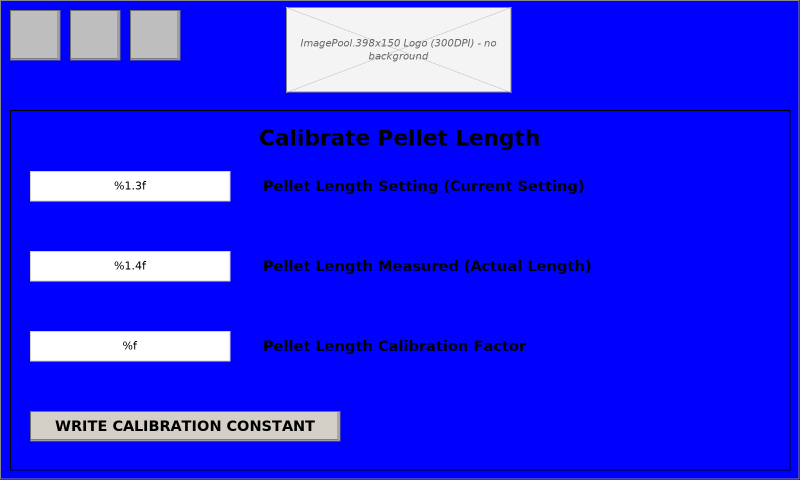
VISUALIZATION Calibrate_Settings  // 800x480
    Rectangle (0,0 800x480)
    Rectangle (10,110 780x360)
    Textfield (30,171 200x30), "%1.3f", text variable: GVL.Pellet_Length_Inch_Input
    Textfield (30,251 200x30), "%1.4f", text variable: Pellet_Calibration.Pellet_Length_Measured_Input
        OnMouseClick: write the text variable via VisuDialogs.Numpad
    Textfield (30,331 200x30), "%f", text variable: Pellet_Calibration.Pellet_Length_Temp_Cal_Val
    Image (286,7 225x85), image: ImagePool.398x150 Logo (300DPI) - no background
        OnMouseClick: change screen: Home
    Button (70,10 50x50), image: VisuSymbols.Symbols.Home
        OnMouseClick: change screen: Home
    Label (0,120 800x36), "Calibrate Pellet Length"
    Button (10,10 50x50), image: VisuSymbols.Symbols.TriangleLeft
        OnMouseClick: change screen: Previous Home
    Label (260,171 361x30), "Pellet Length Setting (Current Setting)"
    Label (260,251 421x30), "Pellet Length Measured (Actual Length)"
    Label (260,331 322x30), "Pellet Length Calibration Factor"
    Label (260,411 225x30)
    Label (550,331 225x30)
    Button (30,411 310x30), "WRITE CALIBRATION CONSTANT", pressed state: Pellet_Calibration.SET_CALIBRATON_VALUE
        OnMouseClick: execute { GVL.Pellet_Length_Calibration_Value := Pellet_Calibration.Pellet_Length_Temp_Cal_Val; }
    Button (130,10 50x50), image: VisuSymbols.Symbols.TwoWheels
        OnMouseClick: change screen: Settings_Menu
END_VISUALIZATION

(* stored: Version 1.1.0.1, ProductVersion 3.1.4024.12
   Visu Calibrate_Settings: Id {7cc5e3bf-0ba5-48a9-b628-4a7f56373090} *)
